TYPE ST_ProcessData :
STRUCT
	Batch		: STRING(100);
	DateTime	: DT;
	Value1		: STRING(100);
	Value2		: STRING(100);
	Value3		: STRING(100);
	Value4		: STRING(100);
	Value5		: STRING(100);
	Value6		: STRING(100);
	Value7		: STRING(100);
END_STRUCT
END_TYPE

(* stored: Version 1.1.0.1, ProductVersion 3.1.4024.12
   DUT ST_ProcessData: Id {3d4f24af-b6dc-46ab-9964-91ccef45caf1} *)
